Universal Robots URScript: TesteUFAM.script

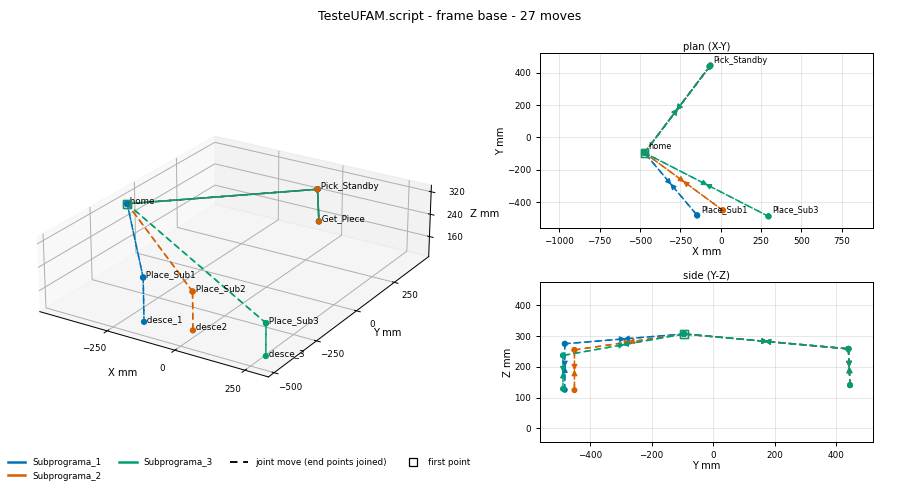
[picture p0: tool path of TesteUFAM.script in frame base, 27 of 27 moves have a stored position in this frame; points joined in program order, loops and branches not executed]
def TesteUFAM():
  set_gravity([0.0, 0.0, 9.82])
  step_count_f0bf7ebe_6968_4ee5_8aa6_65b1d33634db = 0.0
  thread Step_Counter_Thread_8fe2ea37_d722_4b42_96ae_6757ef7a9801():
    while (True):
      step_count_f0bf7ebe_6968_4ee5_8aa6_65b1d33634db = step_count_f0bf7ebe_6968_4ee5_8aa6_65b1d33634db + 1.0
      sync()
    end
  end
  run Step_Counter_Thread_8fe2ea37_d722_4b42_96ae_6757ef7a9801()
  set_tool_voltage(24)
  set_tcp(p[0.0,0.0,0.13,0.0,0.0,0.0])
  set_payload(0.5)
  set_standard_analog_input_domain(0, 1)
  set_standard_analog_input_domain(1, 1)
  set_tool_analog_input_domain(0, 1)
  set_tool_analog_input_domain(1, 1)
  set_analog_outputdomain(0, 0)
  set_analog_outputdomain(1, 0)
  set_input_actions_to_default()
  set_safety_mode_transition_hardness(1)
  global Posicao=[0, 0, 0]
  global Plano_2=p[-0.2971724967048656,0.6250943309952991,0.36888637493592585,-1.0281767974108946,-0.09875334673152589,0.4159429145115416]
  def Subprograma_1():
    $ 16 "Subprograma_1" "noBreak"
    $ 17 "Movimento J"
    $ 18 "home" "breakAfter"
    movej(get_inverse_kin(p[-.472186875617, -.094667915222, .306700472967, 2.140691290721, 2.267434092265, -.061098023954], qnear=[-0.052496735249658144, -1.6228421370135662, 1.613163948059075, -1.5691064039813316, -1.531962219868789, -0.1093595663653808]), a=1.3962634015954636, v=1.0471975511965976)
    $ 19 "Movimento J"
    $ 20 "Pick_Standby" "breakAfter"
    movej(get_inverse_kin(p[-.068331414927, .440444481290, .258292151294, -3.069131651706, .033374410039, .106785363747], qnear=[-1.7040074507342737, -1.7357824484454554, 1.8515729904174805, -1.7479870955096644, -1.499017063771383, -0.10968286195863897]), a=3.490658503988659, v=1.3962634015954636)
    $ 21 "Get_Piece" "breakAfter"
    movej(get_inverse_kin(p[-.063950924512, .445684939631, .140169603666, -3.109069167102, .037734812771, .087367402671], qnear=[-1.7036469618426722, -1.6247146765338343, 2.057220935821533, -2.027203385029928, -1.5167177359210413, -0.10969478288759404]), a=5.235987755982989, v=1.7453292519943295)
    $ 22 "Pick_Standby" "breakAfter"
    movej(get_inverse_kin(p[-.068331414927, .440444481290, .258292151294, -3.069131651706, .033374410039, .106785363747], qnear=[-1.7040074507342737, -1.7357824484454554, 1.8515729904174805, -1.7479870955096644, -1.499017063771383, -0.10968286195863897]), a=5.235987755982989, v=1.3962634015954636)
    $ 23 "Movimento J"
    $ 24 "home" "breakAfter"
    movej(get_inverse_kin(p[-.472186875617, -.094667915222, .306700472967, 2.140691290721, 2.267434092265, -.061098023954], qnear=[-0.052496735249658144, -1.6228421370135662, 1.613163948059075, -1.5691064039813316, -1.531962219868789, -0.1093595663653808]), a=1.3962634015954636, v=1.0471975511965976)
    $ 25 "Movimento J"
    $ 26 "Place_Sub1" "breakAfter"
    movej(get_inverse_kin(p[-.145792539946, -.482461054758, .274899411804, -.617207380519, -3.072180270960, -.042376665246], qnear=[1.0642658472061157, -1.543976132069723, 1.6085233688354492, -1.6118057409869593, -1.5920780340777796, -0.10947925249208623]), a=1.3962634015954636, v=1.0471975511965976)
    $ 27 "desce_1" "breakAfter"
    movej(get_inverse_kin(p[-.145773812690, -.482461927738, .124935837398, -.617180096289, -3.072124846066, -.042277700785], qnear=[1.0643497705459533, -1.452237431203021, 1.9073414802551198, -2.0024741331683416, -1.5918024222003249, -0.1112397352801846]), a=1.3962634015954636, v=1.0471975511965976)
    $ 28 "Place_Sub1" "breakAfter"
    movej(get_inverse_kin(p[-.145792539946, -.482461054758, .274899411804, -.617207380519, -3.072180270960, -.042376665246], qnear=[1.0642658472061157, -1.543976132069723, 1.6085233688354492, -1.6118057409869593, -1.5920780340777796, -0.10947925249208623]), a=1.3962634015954636, v=1.0471975511965976)
    $ 29 "Movimento J"
    $ 30 "home" "breakAfter"
    movej(get_inverse_kin(p[-.472186875617, -.094667915222, .306700472967, 2.140691290721, 2.267434092265, -.061098023954], qnear=[-0.052496735249658144, -1.6228421370135662, 1.613163948059075, -1.5691064039813316, -1.531962219868789, -0.1093595663653808]), a=1.3962634015954636, v=1.0471975511965976)
    $ 31 "Definir DO[5]=Ligar"
    set_standard_digital_out(5, True)
  end
  def Subprograma_2():
    $ 32 "Subprograma_2" "noBreak"
    $ 33 "Movimento J"
    $ 34 "home" "breakAfter"
    movej(get_inverse_kin(p[-.472186875617, -.094667915222, .306700472967, 2.140691290721, 2.267434092265, -.061098023954], qnear=[-0.052496735249658144, -1.6228421370135662, 1.613163948059075, -1.5691064039813316, -1.531962219868789, -0.1093595663653808]), a=1.3962634015954636, v=1.0471975511965976)
    $ 35 "Movimento J"
    $ 36 "Pick_Standby" "breakAfter"
    movej(get_inverse_kin(p[-.068331414927, .440444481290, .258292151294, -3.069131651706, .033374410039, .106785363747], qnear=[-1.7040074507342737, -1.7357824484454554, 1.8515729904174805, -1.7479870955096644, -1.499017063771383, -0.10968286195863897]), a=1.3962634015954636, v=1.0471975511965976)
    $ 37 "Get_Piece" "breakAfter"
    movej(get_inverse_kin(p[-.063950924512, .445684939631, .140169603666, -3.109069167102, .037734812771, .087367402671], qnear=[-1.7036469618426722, -1.6247146765338343, 2.057220935821533, -2.027203385029928, -1.5167177359210413, -0.10969478288759404]), a=1.3962634015954636, v=1.0471975511965976)
    $ 38 "Pick_Standby" "breakAfter"
    movej(get_inverse_kin(p[-.068331414927, .440444481290, .258292151294, -3.069131651706, .033374410039, .106785363747], qnear=[-1.7040074507342737, -1.7357824484454554, 1.8515729904174805, -1.7479870955096644, -1.499017063771383, -0.10968286195863897]), a=1.3962634015954636, v=1.0471975511965976)
    $ 39 "Movimento J"
    $ 40 "home" "breakAfter"
    movej(get_inverse_kin(p[-.472186875617, -.094667915222, .306700472967, 2.140691290721, 2.267434092265, -.061098023954], qnear=[-0.052496735249658144, -1.6228421370135662, 1.613163948059075, -1.5691064039813316, -1.531962219868789, -0.1093595663653808]), a=1.3962634015954636, v=1.0471975511965976)
    $ 41 "Movimento J"
    $ 42 "Place_Sub2" "breakAfter"
    movej(get_inverse_kin(p[.012917010703, -.451008740497, .254716358806, -.161000134099, -3.124454152442, -.015518113325], qnear=[1.3605402708053536, -1.6755855719195738, 1.7899184226989693, -1.677275959645395, -1.590951267872934, -0.10735971132388755]), a=1.3962634015954636, v=1.0471975511965976)
    $ 43 "desce2" "breakAfter"
    movej(get_inverse_kin(p[.012903937211, -.451028262398, .123911944306, -.160855025210, -3.124389506653, -.015445464066], qnear=[1.3605642318725586, -1.5815609137164515, 2.0521111488342285, -2.0335801283465784, -1.5906279722796839, -0.10908395448793584]), a=1.3962634015954636, v=1.0471975511965976)
    $ 44 "Place_Sub2" "breakAfter"
    movej(get_inverse_kin(p[.012917010703, -.451008740497, .254716358806, -.161000134099, -3.124454152442, -.015518113325], qnear=[1.3605402708053536, -1.6755855719195738, 1.7899184226989693, -1.677275959645395, -1.590951267872934, -0.10735971132388755]), a=1.3962634015954636, v=1.0471975511965976)
    $ 45 "Movimento J"
    $ 46 "home" "breakAfter"
    movej(get_inverse_kin(p[-.472186875617, -.094667915222, .306700472967, 2.140691290721, 2.267434092265, -.061098023954], qnear=[-0.052496735249658144, -1.6228421370135662, 1.613163948059075, -1.5691064039813316, -1.531962219868789, -0.1093595663653808]), a=1.3962634015954636, v=1.0471975511965976)
    $ 47 "Definir DO[5]=Ligar"
    set_standard_digital_out(5, True)
  end
  def Subprograma_3():
    $ 48 "Subprograma_3" "noBreak"
    $ 49 "Movimento J"
    $ 50 "home" "breakAfter"
    movej(get_inverse_kin(p[-.472186875617, -.094667915222, .306700472967, 2.140691290721, 2.267434092265, -.061098023954], qnear=[-0.052496735249658144, -1.6228421370135662, 1.613163948059075, -1.5691064039813316, -1.531962219868789, -0.1093595663653808]), a=1.3962634015954636, v=1.0471975511965976, r=0.05)
    $ 51 "Movimento J"
    $ 52 "Pick_Standby" "breakAfter"
    movej(get_inverse_kin(p[-.068331414927, .440444481290, .258292151294, -3.069131651706, .033374410039, .106785363747], qnear=[-1.7040074507342737, -1.7357824484454554, 1.8515729904174805, -1.7479870955096644, -1.499017063771383, -0.10968286195863897]), a=1.3962634015954636, v=1.0471975511965976)
    $ 53 "Get_Piece" "breakAfter"
    movej(get_inverse_kin(p[-.063950924512, .445684939631, .140169603666, -3.109069167102, .037734812771, .087367402671], qnear=[-1.7036469618426722, -1.6247146765338343, 2.057220935821533, -2.027203385029928, -1.5167177359210413, -0.10969478288759404]), a=1.3962634015954636, v=1.0471975511965976)
    $ 54 "Pick_Standby" "breakAfter"
    movej(get_inverse_kin(p[-.068331414927, .440444481290, .258292151294, -3.069131651706, .033374410039, .106785363747], qnear=[-1.7040074507342737, -1.7357824484454554, 1.8515729904174805, -1.7479870955096644, -1.499017063771383, -0.10968286195863897]), a=1.3962634015954636, v=1.0471975511965976)
    $ 55 "Movimento J"
    $ 56 "home" "breakAfter"
    movej(get_inverse_kin(p[-.472186875617, -.094667915222, .306700472967, 2.140691290721, 2.267434092265, -.061098023954], qnear=[-0.052496735249658144, -1.6228421370135662, 1.613163948059075, -1.5691064039813316, -1.531962219868789, -0.1093595663653808]), a=1.3962634015954636, v=1.0471975511965976)
    $ 57 "Movimento J"
    $ 58 "Place_Sub3" "breakAfter"
    movej(get_inverse_kin(p[.295836285148, -.488385197708, .236954256728, -.657003112538, 2.995418860300, -.012015507168], qnear=[1.8936854600906372, -1.4019001165973108, 1.5595555305480957, -1.7441518942462366, -1.5027201811419886, -0.10856897035707647]), a=1.3962634015954636, v=1.0471975511965976)
    $ 59 "desce_3" "breakAfter"
    movej(get_inverse_kin(p[.295842132491, -.488373886106, .128212613212, -.657002192688, 2.995462163162, -.012238457730], qnear=[1.8937333822250366, -1.327808682118551, 1.758786678314209, -2.0175297896014612, -1.5024684111224573, -0.10976678529848272]), a=1.3962634015954636, v=1.0471975511965976)
    $ 60 "Place_Sub3" "breakAfter"
    movej(get_inverse_kin(p[.295836285148, -.488385197708, .236954256728, -.657003112538, 2.995418860300, -.012015507168], qnear=[1.8936854600906372, -1.4019001165973108, 1.5595555305480957, -1.7441518942462366, -1.5027201811419886, -0.10856897035707647]), a=1.3962634015954636, v=1.0471975511965976)
    $ 61 "Movimento J"
    $ 62 "home" "breakAfter"
    movej(get_inverse_kin(p[-.472186875617, -.094667915222, .306700472967, 2.140691290721, 2.267434092265, -.061098023954], qnear=[-0.052496735249658144, -1.6228421370135662, 1.613163948059075, -1.5691064039813316, -1.531962219868789, -0.1093595663653808]), a=1.3962634015954636, v=1.0471975511965976)
    $ 63 "Definir DO[5]=Ligar"
    set_standard_digital_out(5, True)
  end
  def Subprograma_4():
    $ 64 "Subprograma_4" "noBreak"
    $ 65 "Aguardar: 1.0"
    sleep(1.0)
    $ 66 "Definir DO[5]=Desligar"
    set_standard_digital_out(5, False)
    $ 67 "Aguardar: 1.0"
    sleep(1.0)
    $ 68 "Definir DO[0]=Desligar"
    set_standard_digital_out(0, False)
    $ 69 "Aguardar: 1.0"
    sleep(1.0)
    $ 70 "Definir DO[1]=Desligar"
    set_standard_digital_out(1, False)
    $ 71 "Aguardar: 1.0"
    sleep(1.0)
    $ 72 "Definir DO[2]=Desligar"
    set_standard_digital_out(2, False)
  end
  $ 1 "Programa do Robô"
  $ 2 "Loop"
  while (True):
    $ 3 "Aguardar: 1.0"
    sleep(1.0)
    $ 4 "Se digital_out[0] ≟  True  and (digital_out[1] ≟ False  and digital_out[2] ≟ True)"
    if (get_standard_digital_out(0)  ==    True    and  (digital_out[1]  ==  False   and  digital_out[2]  ==  True)):
      $ 5 "Chamar Subprograma_1"
      Subprograma_1()
      $ 6 "Chamar Subprograma_4"
      Subprograma_4()
      $ 7 "Aguardar: 2.0"
      sleep(2.0)
    end
    $ 8 "Se digital_out[0] ≟  True  and (digital_out[1] ≟ True  and digital_out[2] ≟  False )"
    if (get_standard_digital_out(0)  ==    True    and  (digital_out[1]  ==  True   and  digital_out[2]  ==    False  )):
      $ 9 "Chamar Subprograma_2"
      Subprograma_2()
      $ 10 "Chamar Subprograma_4"
      Subprograma_4()
      $ 11 "Aguardar: 2.0"
      sleep(2.0)
    end
    $ 12 "Se digital_out[0] ≟  True  and (digital_out[1] ≟ True  and digital_out[2] ≟ True )"
    if (get_standard_digital_out(0)  ==    True    and  (digital_out[1]  ==  True   and  digital_out[2]  ==   True  )):
      $ 13 "Chamar Subprograma_3"
      Subprograma_3()
      $ 14 "Chamar Subprograma_4"
      Subprograma_4()
      $ 15 "Aguardar: 2.0"
      sleep(2.0)
    end
  end
end
